(* IEC 61131-3 sources: julia_exos_development/src/StringAndArray_JS/StringAndA, 2 files *)

(* ---- StringAndArray.typ ---- *)
TYPE
	IntStruct_typ : 	STRUCT
		MyInt13 : UDINT;
		MyInt14 : ARRAY[0..2]OF USINT;
		MyInt133 : UDINT;
		MyInt124 : ARRAY[0..2]OF USINT;
	END_STRUCT;
	IntStruct1_typ : 	STRUCT
		MyInt13 : UDINT;
	END_STRUCT;
	IntStruct2_typ : 	STRUCT
		MyInt23 : UDINT;
		MyInt24 : ARRAY[0..3]OF USINT;
		MyInt25 : UDINT;
	END_STRUCT;
	StringAndArray : 	STRUCT
		MyInt1 : UDINT; (*PUB*)
		MyString : ARRAY[0..2]OF STRING[80]; (*PUB*)
		MyInt2 : ARRAY[0..4]OF USINT; (*PUB SUB*)
		MyIntStruct : ARRAY[0..5]OF IntStruct_typ; (*PUB SUB*)
		MyIntStruct1 : IntStruct1_typ; (*PUB SUB*)
		MyIntStruct2 : IntStruct2_typ; (*PUB SUB*)
	END_STRUCT;
END_TYPE

(* ---- StringAndA.fun ---- *)
FUNCTION_BLOCK StringAndArrayInit
	VAR_OUTPUT
		Handle : UDINT;
	END_VAR
	VAR
		_state : USINT;
	END_VAR
END_FUNCTION_BLOCK

FUNCTION_BLOCK StringAndArrayCyclic
	VAR_INPUT
		Enable : BOOL;
		Handle : UDINT;
		Start : BOOL;
		pStringAndArray : REFERENCE TO StringAndArray;
	END_VAR
	VAR_OUTPUT
		Active : BOOL;
		Error : BOOL;
		Disconnected : BOOL;
		Connected : BOOL;
		Operational : BOOL;
		Aborted : BOOL;
	END_VAR
	VAR
		_state : USINT;
	END_VAR
END_FUNCTION_BLOCK

FUNCTION_BLOCK StringAndArrayExit
	VAR_INPUT
		Handle : UDINT;
	END_VAR
	VAR
		_state : USINT;
	END_VAR
END_FUNCTION_BLOCK
